// TIA Portal V17 export
// export: Created 2022-07-20T07:02:32.4110836Z, ExportSetting WithDefaults, DisplayName Totally Integrated Automation Portal, DisplayVersion V17, DisplayName TIA Portal Openness, DisplayVersion V17, DisplayName TIA Portal Version Control Interface, DisplayVersion V17, DisplayName SINAMICS Startdrive Advanced, DisplayVersion V17, DisplayName SINAMICS Startdrive G130, G150, S120, S150, SINAMICS MV, S210, DisplayVersion V17, DisplayName SINAMICS Startdrive G110M, G120, G120C, G120D, G120P, G115D, DisplayVersion V17, DisplayName STEP 7 Professional, DisplayVersion V17, DisplayName STEP 7 Safety, DisplayVersion V17, DisplayName WinCC Advanced, DisplayVersion V17
FUNCTION_BLOCK "FB11002_CamTrackConvertProfile"   // FB11002, LAD
TITLE = Transfert and check data of foil profile
{ S7_Optimized_Access := 'TRUE' }
VERSION : 0.1
// stored: AutoNumber false, IsIECCheckEnabled false, IsRetainMemResEnabled false, MemoryReserve 100, SetENOAutomatically false, UDAEnableTagReadback false
   VAR_INPUT
      Execute { ExternalAccessible := 'False'; ExternalVisible := 'False'; ExternalWritable := 'False'} : Bool;
      OffsetGap { ExternalAccessible := 'False'; ExternalVisible := 'False'; ExternalWritable := 'False'} : Real;
      SheetProfile { ExternalAccessible := 'False'; ExternalVisible := 'False'; ExternalWritable := 'False'} : "stSheetProfile";
      StartSheetPosition : LReal;
   END_VAR
   VAR_OUTPUT
      Done { ExternalAccessible := 'False'; ExternalVisible := 'False'; ExternalWritable := 'False'} : Bool;
      Error { ExternalAccessible := 'False'; ExternalVisible := 'False'; ExternalWritable := 'False'} : Bool;
      CamProfile { ExternalAccessible := 'False'; ExternalVisible := 'False'; ExternalWritable := 'False'} : Array[1..32] of TO_CamTrack_Struct_CamData;
   END_VAR
   VAR
      statNumberOfArea : UInt;
      statExecuteOld : Bool;
      statDone : Bool;
      statError : Bool;
      R_TRIG_Execute : R_TRIG;
   END_VAR
   VAR_TEMP
      AreaNumber : UInt;
      segmentNumber : UInt;
      tempTotLength : Real;
   END_VAR
   VAR CONSTANT
      ratioFoilUnwinder : Real := 2.5;
      ratioDeadZone : Real := 1.0;
   END_VAR
   // // SheetProfile.Length : [mm]
BEGIN

REGION Network 1 (SCL): Comments
   //==========================================================================================
   // SIEMENS SAS      RC-FR DI FA APC
   //------------------------------------------------------------------------------------------
   // Restrictions:    TIA V16 and more
   // Requirements:    S7-1500T + MGI library
   // Functionality:   This function block convert stSheetProfile into stCamTrack
   // and check data
   //------------------------------------------------------------------------------------------
   // Change log table:
   // Version      Date        Expert in charge    Changes applied
   // 01.00.01     09.06.2020  RTO                 First released version
   //==========================================================================================
END_REGION

REGION Network 2 (SCL): Edge Signals & Timers
   REGION EDGE SIGNALS
       #R_TRIG_Execute(CLK := #Execute);
   END_REGION
END_REGION

REGION Network 3 (SCL): Manage data
   IF NOT #Execute THEN
       #statDone := FALSE;
       #statError := FALSE;
   END_IF;

   IF #R_TRIG_Execute.Q THEN

       REGION Parameters
           // Get number of area used
           #statNumberOfArea := 0;
           FOR #AreaNumber := 1 TO "MAX_NUMBER_OF_FOIL_AREA" DO
               IF #SheetProfile.Area[#AreaNumber].Start <> #SheetProfile.Area[#AreaNumber].End THEN
                   #statNumberOfArea := #statNumberOfArea + 1;
               END_IF;
           END_FOR;

               // Parameters error
               IF #statNumberOfArea = 0
               THEN
                   #statError := TRUE;
               END_IF;

           // Clear CamProfile
           FOR #segmentNumber := 1 TO 32 DO
               #CamProfile[#segmentNumber].Existent := FALSE;
           END_FOR;

           // Initializr number of segment
           #segmentNumber := 1;

       END_REGION

       IF NOT #statError THEN
           REGION Segment definition

               //--- AREA SEGMENT ---
               FOR #AreaNumber := 1 TO #statNumberOfArea DO

                   //--- SYNCHRONOUS ---
                   #CamProfile[#segmentNumber].Existent := TRUE;
                   #CamProfile[#segmentNumber].OnPosition := #SheetProfile.Area[#AreaNumber].Start + #SheetProfile.StampAreaStartAdjustment + #OffsetGap + #StartSheetPosition;
                   #CamProfile[#segmentNumber].OffPosition := #SheetProfile.Area[#AreaNumber].End + #SheetProfile.StampAreaStartAdjustment + #SheetProfile.StampAreaLengthAdjustement + #OffsetGap + #StartSheetPosition;
                   #segmentNumber := #segmentNumber + 1;

                       // Error first segment
                       IF #CamProfile[#segmentNumber].OffPosition <= #CamProfile[#segmentNumber].OnPosition
                       THEN
                           #statError := TRUE;
                       END_IF;

               END_FOR;
               //--- END AREA SEGMENT ---

            END_REGION
       END_IF;

       #statDone := TRUE;
   END_IF;
END_REGION

REGION Network 4 (SCL): Manage output
   REGION Output
       #Done := #statDone;
       #Error := #statError;
   END_REGION
END_REGION
END_FUNCTION_BLOCK
